// TIA Portal V20 export
TYPE "typeEstopStatus"
// stored: Access Published, IsFailsafeCompliant true, Namespace Safety
   STRUCT
      mainOpEmoPressed : Bool;   // Main OP EMO pressed
      unwinderCenterEmoPressed : Bool;   // Unwinder Center EMO pressed
      jrOutPutEmoPressed : Bool;   // JR Output EMO pressed
      pHmiEmoPressed : Bool;   // PHMI EMO pressed
      ba10EmoPressed : Bool;   // CathodeReelCut EMO Pressed
      ba15EmoPressed : Bool;   // AnodeReelCut EMO Pressed
      ba40EmoPressed : Bool;   // Stacker2 EMO Pressed
      ba60EmoPressed : Bool;   // Inspection EMO Pressed
   END_STRUCT;
END_TYPE
